FUNCTION_BLOCK McMoveAbsoluteProcess EXTENDS BaseMcProcess
VAR_INPUT
	///Arguments to be set, before writing do_request TRUE
	{attribute 'OPC.UA.DA' := '1'}
	set: McMoveAbsoluteProcessArgs;
END_VAR
VAR_OUTPUT
	///Arguments in use by the process, if do_request was accepted
	{attribute 'OPC.UA.DA' := '1'}
	{attribute 'OPC.UA.DA.Access' := '1'}
	get: McMoveAbsoluteProcessArgs;
END_VAR
VAR_IN_OUT
END_VAR
VAR
END_VAR

IF do_request THEN
    do_request_result := request(
    position := set.position,
    maxVelocity := set.maxVelocity);
    do_request := FALSE;
END_IF;
SUPER^();

{attribute 'TcRpcEnable' := '1'}
METHOD request : RequestResults
VAR_INPUT
	///New position setpoint
	position: LREAL;
	///Maximum velocity
	maxVelocity: LREAL;
END_VAR
VAR_OUTPUT
END_VAR
VAR_IN_OUT
END_VAR
VAR
END_VAR
IF THIS^.statuses.enabledStatus.enabled THEN
    THIS^.start(
        position := position,
        maxVelocity := maxVelocity);
    request := RequestResults.ACCEPTED;
ELSE
    request := RequestResults.REJECTED;
END_IF;
END_METHOD

{attribute 'TcRpcEnable' := '1'}
METHOD start
VAR_INPUT
	///New position setpoint
	position: LREAL;
	///Maximum velocity
	maxVelocity: LREAL;
END_VAR
VAR_OUTPUT
END_VAR
VAR_IN_OUT
END_VAR
VAR
END_VAR
THIS^.get.position := position;
THIS^.get.maxVelocity := maxVelocity;
THIS^.statuses.busyStatus( isBusy := TRUE );
THIS^.statuses.healthStatus( isGood := TRUE );
END_METHOD

END_FUNCTION_BLOCK

(* stored: Version 1.1.0.1, ProductVersion 3.1.4019.2
   POU McMoveAbsoluteProcess: Id {48af296d-f77e-42c9-90aa-141e92b63b53}, SpecialFunc None
   Method request: Id {9b847641-4688-402e-aefb-5eab76b64525}
   Method start: Id {c621e88c-a00f-4005-a360-e89fdf2da08c} *)
